Universal Robots PolyScope program: Assem_SubAssem1.urp

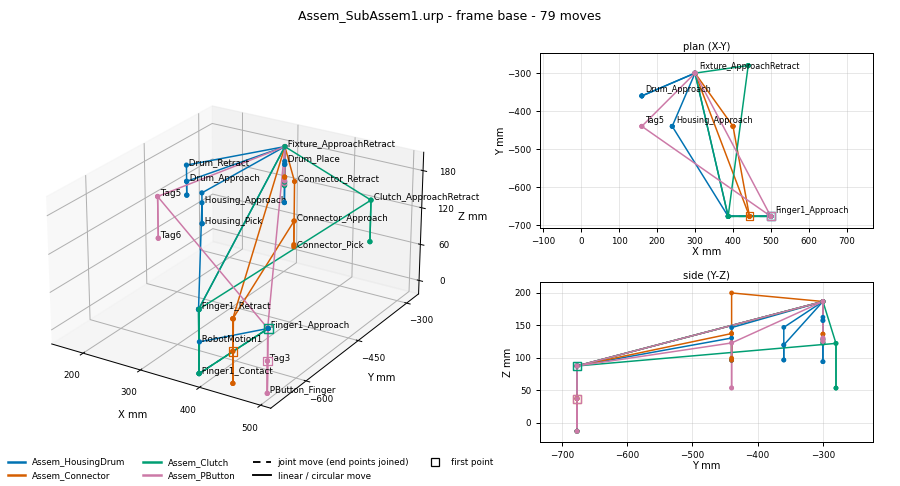
[picture p0: tool path of Assem_SubAssem1.urp in frame base, 79 of 79 moves have a stored position in this frame; points joined in program order, loops and branches not executed]
Program Assem_SubAssem1 (createdIn=3.7.2.40245 lastSavedIn=3.7.2.40245 robotSerialNumber= directory= installation=)
Robot Program (runOnlyOnce=false)
  Call Assem_HousingDrum
  Call Assem_Connector
  Call Assem_Clutch
  Call Assem_PButton
SubProgram -> Assem_HousingDrum
SubProgram -> Assem_Connector
SubProgram -> Assem_Clutch
SubProgram -> Assem_PButton
SubProgram Assem_HousingDrum (keepSynchronizedWithDisk=false trackProgramExecution=true)
  MoveJ speed 120 deg/s, acceleration 360 deg/s^2 (useActiveTCP=false) tcp=TCP_1; feature=Base
    Waypoint Finger1_Approach: TCP in base x=500.448 y=-677.024 z=87.412 mm, rx=-2.2214 ry=2.2214 rz=0 rad; joints [-44.419, -144.242, -45.363, -80.394, 90, -44.419] deg; flange x=500.447 y=-677.022 z=245.817 mm, rx=-2.2214 ry=2.2214 rz=0 rad
  Script: rq_activate_and_wait()
  URCap Gripper (Robotiq_Grippers, Robotiq Inc.) dataModel(position=25, force=50, speed=50, blocking=true, positionInDouble=25.0, forceInDouble=50.0, speedInDouble=50.0)
  MoveL speed 250 mm/s, acceleration 5000 mm/s^2 (useActiveTCP=false) tcp=TCP_1; feature=Base
    Waypoint RobotMotion1: TCP in base x=388.248 y=-677.024 z=37.407 mm, rx=2.2214 ry=-2.2214 rz=0 rad; joints [-50.333, -136.868, -66.833, -66.298, 90, -50.333] deg; flange x=388.247 y=-677.023 z=195.812 mm, rx=2.2214 ry=-2.2214 rz=0 rad
  Set DigitalOutput pin=config_out[0]; digitalValue=1
  MoveL speed 250 mm/s, acceleration 5000 mm/s^2 (useActiveTCP=false) tcp=TCP_1; feature=Base
    Waypoint Finger1_Contact: TCP in base x=387.249 y=-677.025 z=-12.589 mm, rx=-2.2214 ry=2.2214 rz=-0.0001 rad; joints [-50.391, -140.03, -68.963, -61.003, 90, -50.39] deg; flange x=387.242 y=-677.017 z=145.816 mm, rx=-2.2214 ry=2.2214 rz=-0.0001 rad
  Set DigitalOutput pin=config_out[0]; digitalValue=0
  Wait Sleep waitTime=1
  MoveL speed 250 mm/s, acceleration 5000 mm/s^2 (useActiveTCP=false) tcp=TCP_1; feature=Base
    Waypoint Finger1_Retract: TCP in base x=387.248 y=-677.024 z=87.414 mm, rx=-2.2214 ry=2.2214 rz=0 rad; joints [-50.39, -134.151, -63.976, -71.872, 90, -50.39] deg; flange x=387.246 y=-677.022 z=245.819 mm, rx=-2.2214 ry=2.2214 rz=0 rad
  MoveL speed 250 mm/s, acceleration 5000 mm/s^2 (useActiveTCP=false) tcp=TCP_1; feature=Base
    Waypoint Housing_Approach: TCP in base x=240 y=-440 z=130.253 mm, rx=2.2214 ry=-2.2214 rz=0 rad; joints [-45.965, -95.978, -114.162, -59.858, 90, -45.965] deg; flange x=239.997 y=-439.996 z=288.658 mm, rx=2.2214 ry=-2.2214 rz=0 rad
  MoveL speed 250 mm/s, acceleration 5000 mm/s^2 (useActiveTCP=false) tcp=TCP_1; feature=Base
    Waypoint Housing_Pick: TCP in base x=240 y=-440 z=96.255 mm, rx=-2.2214 ry=2.2214 rz=-0.0001 rad; joints [-45.965, -98.735, -116.867, -54.395, 90, -45.965] deg; flange x=239.994 y=-439.994 z=254.66 mm, rx=-2.2214 ry=2.2214 rz=-0.0001 rad
  URCap Gripper (Robotiq_Grippers, Robotiq Inc.) dataModel(position=80, force=50, speed=50, blocking=true, positionInDouble=80.0, forceInDouble=50.0, speedInDouble=50.0)
  MoveL speed 250 mm/s, acceleration 5000 mm/s^2 (useActiveTCP=false) tcp=TCP_1; feature=Base
    Waypoint RobotMotion2: TCP in base x=240 y=-440 z=96.257 mm, rx=2.2214 ry=-2.2214 rz=0.0001 rad; joints [-45.965, -98.735, -116.866, -54.397, 90, -45.965] deg; flange x=239.996 y=-439.995 z=254.662 mm, rx=2.2214 ry=-2.2214 rz=0.0001 rad
  MoveL speed 250 mm/s, acceleration 5000 mm/s^2 (useActiveTCP=false) tcp=TCP_1; feature=Base
    Waypoint Housing_Retract: TCP in base x=240 y=-439.999 z=146.257 mm, rx=2.2214 ry=-2.2214 rz=0.0001 rad; joints [-45.965, -94.842, -112.761, -62.393, 90, -45.965] deg; flange x=239.994 y=-439.993 z=304.662 mm, rx=2.2214 ry=-2.2214 rz=0.0001 rad
  MoveL speed 250 mm/s, acceleration 5000 mm/s^2 (useActiveTCP=false) tcp=TCP_1; feature=Base
    Waypoint Fixture_ApproachRetract: TCP in base x=299.997 y=-299.998 z=186.263 mm, rx=-2.2214 ry=2.2214 rz=-0.0002 rad; joints [-26.687, -81.35, -119.315, -69.329, 89.999, -26.687] deg; flange x=299.983 y=-299.987 z=344.668 mm, rx=-2.2214 ry=2.2214 rz=-0.0002 rad
  MoveL speed 250 mm/s, acceleration 5000 mm/s^2 (useActiveTCP=false) tcp=TCP_1; feature=Base
    Waypoint Housing_Place: TCP in base x=300 y=-300 z=94.01 mm, rx=-2.2214 ry=2.2214 rz=-0.0001 rad; joints [-26.687, -88.56, -128.317, -53.117, 89.999, -26.687] deg; flange x=299.989 y=-299.991 z=252.415 mm, rx=-2.2214 ry=2.2214 rz=-0.0001 rad
  URCap Gripper (Robotiq_Grippers, Robotiq Inc.) dataModel(position=25, force=50, speed=50, blocking=true, positionInDouble=25.0, forceInDouble=50.0, speedInDouble=50.0)
  MoveL speed 250 mm/s, acceleration 5000 mm/s^2 (useActiveTCP=false) tcp=TCP_1; feature=Base
    Waypoint RobotMotion3: TCP in base x=300.001 y=-300 z=94.012 mm, rx=-2.2214 ry=2.2214 rz=-0.0002 rad; joints [-26.687, -88.56, -128.317, -53.117, 89.999, -26.687] deg; flange x=299.988 y=-299.991 z=252.417 mm, rx=-2.2214 ry=2.2214 rz=-0.0002 rad
  MoveL speed 250 mm/s, acceleration 5000 mm/s^2 (useActiveTCP=false) tcp=TCP_1; feature=Base
    Waypoint Fixture_ApproachRetract: TCP in base x=299.997 y=-299.998 z=186.263 mm, rx=-2.2214 ry=2.2214 rz=-0.0002 rad; joints [-26.687, -81.35, -119.315, -69.329, 89.999, -26.687] deg; flange x=299.983 y=-299.987 z=344.668 mm, rx=-2.2214 ry=2.2214 rz=-0.0002 rad
  MoveL speed 250 mm/s, acceleration 5000 mm/s^2 (useActiveTCP=false) tcp=TCP_1; feature=Base
    Waypoint Drum_Approach: TCP in base x=160 y=-360 z=119.602 mm, rx=-2.2214 ry=2.2214 rz=-0.0002 rad; joints [-46.261, -81.439, -130.102, -58.452, 90.001, -46.261] deg; flange x=159.987 y=-359.99 z=278.007 mm, rx=-2.2214 ry=2.2214 rz=-0.0002 rad
  URCap Gripper (Robotiq_Grippers, Robotiq Inc.) dataModel(position=100, force=50, speed=50, blocking=true, positionInDouble=100.0, forceInDouble=50.0, speedInDouble=50.0)
  MoveL speed 250 mm/s, acceleration 5000 mm/s^2 (useActiveTCP=false) tcp=TCP_1; feature=Base
    Waypoint RobotMotion4: TCP in base x=160 y=-360 z=119.604 mm, rx=-2.2214 ry=2.2214 rz=0 rad; joints [-46.26, -81.442, -130.099, -58.459, 90, -46.26] deg; flange x=159.999 y=-359.999 z=278.009 mm, rx=-2.2214 ry=2.2214 rz=0 rad
  MoveL speed 250 mm/s, acceleration 5000 mm/s^2 (useActiveTCP=false) tcp=TCP_1; feature=Base
    Waypoint Drum_Pick: TCP in base x=160 y=-360 z=96.603 mm, rx=-2.2214 ry=2.2214 rz=0 rad; joints [-46.26, -83.73, -132.237, -54.031, 90, -46.26] deg; flange x=159.999 y=-359.999 z=255.008 mm, rx=-2.2214 ry=2.2214 rz=0 rad
  URCap Gripper (Robotiq_Grippers, Robotiq Inc.) dataModel(position=90, force=50, speed=50, blocking=true, positionInDouble=90.0, forceInDouble=50.0, speedInDouble=50.0)
  MoveL speed 250 mm/s, acceleration 5000 mm/s^2 (useActiveTCP=false) tcp=TCP_1; feature=Base
    Waypoint RobotMotion5: TCP in base x=160 y=-360 z=96.605 mm, rx=-2.2214 ry=2.2214 rz=0 rad; joints [-46.26, -83.73, -132.237, -54.031, 90, -46.26] deg; flange x=159.998 y=-359.998 z=255.01 mm, rx=-2.2214 ry=2.2214 rz=0 rad
  MoveL speed 250 mm/s, acceleration 5000 mm/s^2 (useActiveTCP=false) tcp=TCP_1; feature=Base
    Waypoint Drum_Retract: TCP in base x=160 y=-360 z=146.603 mm, rx=-2.2214 ry=2.2214 rz=0 rad; joints [-46.26, -79.175, -127.379, -63.445, 90, -46.26] deg; flange x=159.998 y=-359.998 z=305.008 mm, rx=-2.2214 ry=2.2214 rz=0 rad
  MoveL speed 250 mm/s, acceleration 5000 mm/s^2 (useActiveTCP=false) tcp=TCP_1; feature=Base
    Waypoint Fixture_ApproachRetract: TCP in base x=299.997 y=-299.998 z=186.263 mm, rx=-2.2214 ry=2.2214 rz=-0.0002 rad; joints [-26.687, -81.35, -119.315, -69.329, 89.999, -26.687] deg; flange x=299.983 y=-299.987 z=344.668 mm, rx=-2.2214 ry=2.2214 rz=-0.0002 rad
  MoveL speed 250 mm/s, acceleration 5000 mm/s^2 (useActiveTCP=false) tcp=TCP_1; feature=Base
    Waypoint Drum_Align: TCP in base x=299.997 y=-299.998 z=186.263 mm, rx=1.0745 ry=-2.9521 rz=0.0002 rad; joints [-26.684, -81.35, -119.314, -69.332, 89.995, 23.316] deg; flange x=299.996 y=-299.98 z=344.668 mm, rx=1.0745 ry=-2.9521 rz=0.0002 rad
  MoveL speed 250 mm/s, acceleration 5000 mm/s^2 (useActiveTCP=false) tcp=TCP_1; feature=Base
    Waypoint Drum_Place: TCP in base x=300 y=-300 z=162.113 mm, rx=-1.0745 ry=2.9521 rz=0 rad; joints [-26.688, -82.813, -121.912, -65.274, 90, 23.312] deg; flange x=299.998 y=-299.999 z=320.518 mm, rx=-1.0745 ry=2.9521 rz=0 rad
  MoveL speed 250 mm/s, acceleration 5000 mm/s^2 (useActiveTCP=false) tcp=TCP_1; feature=Base
    Waypoint Drum_Insert: TCP in base x=300 y=-300 z=157.114 mm, rx=3.0671 ry=0.68 rz=0 rad; joints [-26.688, -83.151, -122.43, -64.418, 90, -141.688] deg; flange x=299.997 y=-299.999 z=315.519 mm, rx=3.0671 ry=0.68 rz=0 rad
  URCap Gripper (Robotiq_Grippers, Robotiq Inc.) dataModel(position=100, force=50, speed=50, blocking=true, positionInDouble=100.0, forceInDouble=50.0, speedInDouble=50.0)
  MoveL speed 250 mm/s, acceleration 5000 mm/s^2 (useActiveTCP=false) tcp=TCP_1; feature=Base
    Waypoint RobotMotion6: TCP in base x=299.999 y=-299.999 z=157.115 mm, rx=3.0671 ry=0.68 rz=0 rad; joints [-26.688, -83.151, -122.43, -64.418, 90, -141.688] deg; flange x=299.997 y=-299.998 z=315.52 mm, rx=3.0671 ry=0.68 rz=0 rad
  MoveL speed 250 mm/s, acceleration 5000 mm/s^2 (useActiveTCP=false) tcp=TCP_1; feature=Base
    Waypoint Fixture_ApproachRetract: TCP in base x=299.997 y=-299.998 z=186.263 mm, rx=-2.2214 ry=2.2214 rz=-0.0002 rad; joints [-26.687, -81.35, -119.315, -69.329, 89.999, -26.687] deg; flange x=299.983 y=-299.987 z=344.668 mm, rx=-2.2214 ry=2.2214 rz=-0.0002 rad
  MoveL speed 250 mm/s, acceleration 5000 mm/s^2 (useActiveTCP=false) tcp=TCP_1; feature=Base
    Waypoint Finger1_Retract: TCP in base x=387.248 y=-677.024 z=87.414 mm, rx=-2.2214 ry=2.2214 rz=0 rad; joints [-50.39, -134.151, -63.976, -71.872, 90, -50.39] deg; flange x=387.246 y=-677.022 z=245.819 mm, rx=-2.2214 ry=2.2214 rz=0 rad
  URCap Gripper (Robotiq_Grippers, Robotiq Inc.) dataModel(position=25, force=50, speed=50, blocking=true, positionInDouble=25.0, forceInDouble=50.0, speedInDouble=50.0)
  MoveL speed 250 mm/s, acceleration 5000 mm/s^2 (useActiveTCP=false) tcp=TCP_1; feature=Base
    Waypoint RobotMotion7: TCP in base x=388.249 y=-677.024 z=87.418 mm, rx=2.2214 ry=-2.2214 rz=0 rad; joints [-50.333, -134.223, -63.846, -71.929, 90, -50.333] deg; flange x=388.246 y=-677.022 z=245.823 mm, rx=2.2214 ry=-2.2214 rz=0 rad
  MoveL speed 250 mm/s, acceleration 5000 mm/s^2 (useActiveTCP=false) tcp=TCP_1; feature=Base
    Waypoint Finger1_Contact: TCP in base x=387.249 y=-677.025 z=-12.589 mm, rx=-2.2214 ry=2.2214 rz=-0.0001 rad; joints [-50.391, -140.03, -68.963, -61.003, 90, -50.39] deg; flange x=387.242 y=-677.017 z=145.816 mm, rx=-2.2214 ry=2.2214 rz=-0.0001 rad
  Set DigitalOutput pin=config_out[0]; digitalValue=1
  Wait Sleep waitTime=1
  MoveJ speed 120 deg/s, acceleration 360 deg/s^2 (useActiveTCP=false) tcp=TCP_1; feature=Base
    Waypoint Finger1_Approach: TCP in base x=500.448 y=-677.024 z=87.412 mm, rx=-2.2214 ry=2.2214 rz=0 rad; joints [-44.419, -144.242, -45.363, -80.394, 90, -44.419] deg; flange x=500.447 y=-677.022 z=245.817 mm, rx=-2.2214 ry=2.2214 rz=0 rad
SubProgram Assem_Connector (keepSynchronizedWithDisk=false trackProgramExecution=true)
  MoveL speed 250 mm/s, acceleration 5000 mm/s^2 (useActiveTCP=false) tcp=TCP_1; feature=Base
    Waypoint Finger2_Approach: TCP in base x=443.348 y=-677.023 z=37.402 mm, rx=-2.2214 ry=2.2214 rz=0 rad; joints [-47.301, -140.975, -59.111, -69.913, 90, -47.301] deg; flange x=443.348 y=-677.023 z=195.807 mm, rx=-2.2214 ry=2.2214 rz=0 rad
  MoveL speed 250 mm/s, acceleration 5000 mm/s^2 (useActiveTCP=false) tcp=TCP_1; feature=Base
    Waypoint Finger2_Contact: TCP in base x=443.348 y=-677.023 z=-12.6 mm, rx=2.2214 ry=-2.2214 rz=0 rad; joints [-47.3, -143.968, -61.249, -64.783, 90, -47.3] deg; flange x=443.348 y=-677.023 z=145.805 mm, rx=2.2214 ry=-2.2214 rz=0 rad
  Set DigitalOutput pin=config_out[0]; digitalValue=0
  Wait Sleep waitTime=1
  MoveL speed 250 mm/s, acceleration 5000 mm/s^2 (useActiveTCP=false) tcp=TCP_1; feature=Base
    Waypoint Finger2_Retract: TCP in base x=443.347 y=-677.023 z=87.404 mm, rx=-2.2214 ry=2.2214 rz=0 rad; joints [-47.301, -138.599, -55.894, -75.506, 90, -47.301] deg; flange x=443.346 y=-677.022 z=245.809 mm, rx=-2.2214 ry=2.2214 rz=0 rad
  MoveL speed 250 mm/s, acceleration 5000 mm/s^2 (useActiveTCP=false) tcp=TCP_1; feature=Base
    Waypoint Connector_Approach: TCP in base x=400 y=-440 z=137.121 mm, rx=-2.2214 ry=2.2214 rz=0 rad; joints [-34.772, -133.787, -57.117, 100.904, -90, 145.228] deg; flange x=400 y=-440 z=295.526 mm, rx=-2.2214 ry=2.2214 rz=0 rad
  MoveL speed 250 mm/s, acceleration 5000 mm/s^2 (useActiveTCP=false) tcp=TCP_1; feature=Base
    Waypoint RobotMotion1: TCP in base x=400 y=-440 z=137.127 mm, rx=-2.2214 ry=2.2214 rz=0 rad; joints [-34.772, -133.786, -57.117, 100.904, -90, 145.228] deg; flange x=399.998 y=-439.999 z=295.532 mm, rx=-2.2214 ry=2.2214 rz=0 rad
  MoveL speed 250 mm/s, acceleration 5000 mm/s^2 (useActiveTCP=false) tcp=TCP_1; feature=Base
    Waypoint Connector_Pick: TCP in base x=400 y=-440 z=96.11 mm, rx=-2.2214 ry=2.2214 rz=0 rad; joints [-34.772, -135.283, -60.612, 105.896, -90, 145.228] deg; flange x=399.999 y=-439.999 z=254.515 mm, rx=-2.2214 ry=2.2214 rz=0 rad
  URCap Gripper (Robotiq_Grippers, Robotiq Inc.) dataModel(position=85, force=50, speed=50, blocking=true, positionInDouble=85.0, forceInDouble=50.0, speedInDouble=50.0)
  MoveL speed 250 mm/s, acceleration 5000 mm/s^2 (useActiveTCP=false) tcp=TCP_1; feature=Base
    Waypoint RobotMotion2: TCP in base x=400.001 y=-440 z=99.381 mm, rx=-2.2214 ry=2.2214 rz=0 rad; joints [-34.772, -135.146, -60.363, 105.51, -90, 145.228] deg; flange x=399.998 y=-439.998 z=257.786 mm, rx=-2.2214 ry=2.2214 rz=0 rad
  MoveL speed 250 mm/s, acceleration 5000 mm/s^2 (useActiveTCP=false) tcp=TCP_1; feature=Base
    Waypoint Connector_Retract: TCP in base x=399.999 y=-439.999 z=199.381 mm, rx=-2.2214 ry=2.2214 rz=0 rad; joints [-34.772, -132.555, -50.102, 92.658, -90, 145.228] deg; flange x=399.996 y=-439.997 z=357.786 mm, rx=-2.2214 ry=2.2214 rz=0 rad
  MoveL speed 250 mm/s, acceleration 5000 mm/s^2 (useActiveTCP=false) tcp=TCP_1; feature=Base
    Waypoint Fixture_ApproachRetract: TCP in base x=299.997 y=-299.998 z=186.263 mm, rx=-2.2214 ry=2.2214 rz=-0.0002 rad; joints [-26.687, -107.809, -90.446, 108.261, -89.999, 153.313] deg; flange x=299.983 y=-299.987 z=344.668 mm, rx=-2.2214 ry=2.2214 rz=-0.0002 rad
  MoveL speed 250 mm/s, acceleration 5000 mm/s^2 (useActiveTCP=false) tcp=TCP_1; feature=Base
    Waypoint Connector_Place: TCP in base x=300.002 y=-300.001 z=136.264 mm, rx=-2.2214 ry=2.2214 rz=-0.0002 rad; joints [-26.687, -110.306, -94.864, 115.177, -89.999, 153.313] deg; flange x=299.987 y=-299.99 z=294.669 mm, rx=-2.2214 ry=2.2214 rz=-0.0002 rad
  URCap Gripper (Robotiq_Grippers, Robotiq Inc.) dataModel(position=100, force=50, speed=50, blocking=true, positionInDouble=100.0, forceInDouble=50.0, speedInDouble=50.0)
  MoveL speed 250 mm/s, acceleration 5000 mm/s^2 (useActiveTCP=false) tcp=TCP_1; feature=Base
    Waypoint RobotMotion3: TCP in base x=300.002 y=-300.001 z=136.267 mm, rx=-2.2214 ry=2.2214 rz=-0.0002 rad; joints [-26.687, -110.305, -94.864, 115.177, -89.999, 153.313] deg; flange x=299.986 y=-299.989 z=294.672 mm, rx=-2.2214 ry=2.2214 rz=-0.0002 rad
  MoveL speed 250 mm/s, acceleration 5000 mm/s^2 (useActiveTCP=false) tcp=TCP_1; feature=Base
    Waypoint Fixture_ApproachRetract: TCP in base x=299.997 y=-299.998 z=186.263 mm, rx=-2.2214 ry=2.2214 rz=-0.0002 rad; joints [-26.687, -107.809, -90.446, 108.261, -89.999, 153.313] deg; flange x=299.983 y=-299.987 z=344.668 mm, rx=-2.2214 ry=2.2214 rz=-0.0002 rad
  MoveL speed 250 mm/s, acceleration 5000 mm/s^2 (useActiveTCP=false) tcp=TCP_1; feature=Base
    Waypoint Finger2_Retract: TCP in base x=443.347 y=-677.023 z=87.404 mm, rx=-2.2214 ry=2.2214 rz=0 rad; joints [0, 0, 0, 0, 0, 0] deg; flange x=443.346 y=-677.022 z=245.809 mm, rx=-2.2214 ry=2.2214 rz=0 rad
  URCap Gripper (Robotiq_Grippers, Robotiq Inc.) dataModel(position=25, force=50, speed=50, blocking=true, positionInDouble=25.0, forceInDouble=50.0, speedInDouble=50.0)
  MoveL speed 250 mm/s, acceleration 5000 mm/s^2 (useActiveTCP=false) tcp=TCP_1; feature=Base
    Waypoint RobotMotion4: TCP in base x=444.348 y=-677.023 z=87.407 mm, rx=-2.2214 ry=2.2214 rz=0 rad; joints [0, 0, 0, 0, 0, 0] deg; flange x=444.346 y=-677.022 z=245.812 mm, rx=-2.2214 ry=2.2214 rz=0 rad
  MoveL speed 250 mm/s, acceleration 5000 mm/s^2 (useActiveTCP=false) tcp=TCP_1; feature=Base
    Waypoint Finger2_Contact: TCP in base x=443.348 y=-677.023 z=-12.6 mm, rx=2.2214 ry=-2.2214 rz=0 rad; joints [0, 0, 0, 0, 0, 0] deg; flange x=443.348 y=-677.023 z=145.805 mm, rx=2.2214 ry=-2.2214 rz=0 rad
  Set DigitalOutput pin=config_out[0]; digitalValue=1
  Wait Sleep waitTime=1
  MoveL speed 250 mm/s, acceleration 5000 mm/s^2 (useActiveTCP=false) tcp=TCP_1; feature=Base
    Waypoint Finger2_Approach: TCP in base x=443.348 y=-677.023 z=37.402 mm, rx=-2.2214 ry=2.2214 rz=0 rad; joints [0, 0, 0, 0, 0, 0] deg; flange x=443.348 y=-677.023 z=195.807 mm, rx=-2.2214 ry=2.2214 rz=0 rad
SubProgram Assem_Clutch (keepSynchronizedWithDisk=false trackProgramExecution=true)
  MoveL speed 250 mm/s, acceleration 5000 mm/s^2 (useActiveTCP=false) tcp=TCP_1; feature=Base
    Waypoint Finger1_Approach: TCP in base x=500.448 y=-677.024 z=87.412 mm, rx=-2.2214 ry=2.2214 rz=0 rad; joints [0, 0, 0, 0, 0, 0] deg; flange x=500.447 y=-677.022 z=245.817 mm, rx=-2.2214 ry=2.2214 rz=0 rad
  MoveL speed 250 mm/s, acceleration 5000 mm/s^2 (useActiveTCP=false) tcp=TCP_1; feature=Base
    Waypoint Finger1_Contact: TCP in base x=387.249 y=-677.025 z=-12.589 mm, rx=-2.2214 ry=2.2214 rz=-0.0001 rad; joints [0, 0, 0, 0, 0, 0] deg; flange x=387.242 y=-677.017 z=145.816 mm, rx=-2.2214 ry=2.2214 rz=-0.0001 rad
  Set DigitalOutput pin=config_out[0]; digitalValue=0
  Wait Sleep waitTime=1
  MoveL speed 250 mm/s, acceleration 5000 mm/s^2 (useActiveTCP=false) tcp=TCP_1; feature=Base
    Waypoint Finger1_Retract: TCP in base x=387.248 y=-677.024 z=87.414 mm, rx=-2.2214 ry=2.2214 rz=0 rad; joints [0, 0, 0, 0, 0, 0] deg; flange x=387.246 y=-677.022 z=245.819 mm, rx=-2.2214 ry=2.2214 rz=0 rad
  MoveL speed 250 mm/s, acceleration 5000 mm/s^2 (useActiveTCP=false) tcp=TCP_1; feature=Base
    Waypoint Clutch_ApproachRetract: TCP in base x=440 y=-280 z=122.051 mm, rx=-2.2214 ry=2.2214 rz=0 rad; joints [-17.663, -123.732, -76.54, 110.273, -90, 162.337] deg; flange x=440 y=-280 z=280.456 mm, rx=-2.2214 ry=2.2214 rz=0 rad
  MoveL speed 250 mm/s, acceleration 5000 mm/s^2 (useActiveTCP=false) tcp=TCP_1; feature=Base
    Waypoint Clutch_Pick: TCP in base x=440 y=-280 z=53.553 mm, rx=-2.2214 ry=2.2214 rz=0 rad; joints [-17.663, -127.625, -80.942, 118.568, -90, 162.337] deg; flange x=440 y=-280 z=211.958 mm, rx=-2.2214 ry=2.2214 rz=0 rad
  URCap Gripper (Robotiq_Grippers, Robotiq Inc.) dataModel(position=88, force=50, speed=50, blocking=true, positionInDouble=88.0, forceInDouble=50.0, speedInDouble=50.0)
  MoveL speed 250 mm/s, acceleration 5000 mm/s^2 (useActiveTCP=false) tcp=TCP_1; feature=Base
    Waypoint RobotMotion1: TCP in base x=440 y=-280 z=53.554 mm, rx=-2.2214 ry=2.2214 rz=0 rad; joints [-17.663, -127.625, -80.942, 118.568, -90, 162.337] deg; flange x=439.999 y=-280 z=211.959 mm, rx=-2.2214 ry=2.2214 rz=0 rad
  MoveL speed 250 mm/s, acceleration 5000 mm/s^2 (useActiveTCP=false) tcp=TCP_1; feature=Base
    Waypoint Clutch_ApproachRetract: TCP in base x=440 y=-280 z=122.051 mm, rx=-2.2214 ry=2.2214 rz=0 rad; joints [-17.663, -123.732, -76.54, 110.273, -90, 162.337] deg; flange x=440 y=-280 z=280.456 mm, rx=-2.2214 ry=2.2214 rz=0 rad
  MoveL speed 250 mm/s, acceleration 5000 mm/s^2 (useActiveTCP=false) tcp=TCP_1; feature=Base
    Waypoint Fixture_ApproachRetract: TCP in base x=299.997 y=-299.998 z=186.263 mm, rx=-2.2214 ry=2.2214 rz=-0.0002 rad; joints [-26.687, -107.809, -90.446, 108.261, -89.999, 153.313] deg; flange x=299.983 y=-299.987 z=344.668 mm, rx=-2.2214 ry=2.2214 rz=-0.0002 rad
  MoveL speed 250 mm/s, acceleration 5000 mm/s^2 (useActiveTCP=false) tcp=TCP_1; feature=Base
    Waypoint Clutch_Place: TCP in base x=300.003 y=-300.002 z=123.266 mm, rx=-2.2214 ry=2.2214 rz=-0.0002 rad; joints [-26.687, -111.079, -95.875, 116.961, -89.999, 153.313] deg; flange x=299.987 y=-299.99 z=281.671 mm, rx=-2.2214 ry=2.2214 rz=-0.0002 rad
  URCap Gripper (Robotiq_Grippers, Robotiq Inc.) dataModel(position=75, force=50, speed=50, blocking=true, positionInDouble=75.0, forceInDouble=50.0, speedInDouble=50.0)
  MoveL speed 250 mm/s, acceleration 5000 mm/s^2 (useActiveTCP=false) tcp=TCP_1; feature=Base
    Waypoint RobotMotion2: TCP in base x=300.003 y=-300.002 z=123.267 mm, rx=-2.2214 ry=2.2214 rz=-0.0002 rad; joints [-26.687, -111.079, -95.875, 116.961, -89.999, 153.313] deg; flange x=299.987 y=-299.99 z=281.672 mm, rx=-2.2214 ry=2.2214 rz=-0.0002 rad
  MoveL speed 250 mm/s, acceleration 5000 mm/s^2 (useActiveTCP=false) tcp=TCP_1; feature=Base
    Waypoint Clutch_PushRetract: TCP in base x=300.003 y=-300.001 z=128.267 mm, rx=-2.2214 ry=2.2214 rz=-0.0002 rad; joints [-26.687, -110.776, -95.493, 116.276, -89.999, 153.313] deg; flange x=299.987 y=-299.99 z=286.672 mm, rx=-2.2214 ry=2.2214 rz=-0.0002 rad
  URCap Gripper (Robotiq_Grippers, Robotiq Inc.) dataModel(position=100, force=50, speed=50, blocking=true, positionInDouble=100.0, forceInDouble=50.0, speedInDouble=50.0)
  MoveL speed 250 mm/s, acceleration 5000 mm/s^2 (useActiveTCP=false) tcp=TCP_1; feature=Base
    Waypoint RobotMotion3: TCP in base x=300.003 y=-300.001 z=128.268 mm, rx=-2.2214 ry=2.2214 rz=-0.0002 rad; joints [-26.687, -110.775, -95.493, 116.276, -89.999, 153.313] deg; flange x=299.986 y=-299.99 z=286.673 mm, rx=-2.2214 ry=2.2214 rz=-0.0002 rad
  MoveL speed 250 mm/s, acceleration 5000 mm/s^2 (useActiveTCP=false) tcp=TCP_1; feature=Base
    Waypoint Clutch_Push: TCP in base x=300.003 y=-300.002 z=122.11 mm, rx=-2.2214 ry=2.2214 rz=-0.0002 rad; joints [-26.687, -111.15, -95.962, 117.12, -89.999, 153.313] deg; flange x=299.987 y=-299.99 z=280.515 mm, rx=-2.2214 ry=2.2214 rz=-0.0002 rad
  MoveL speed 250 mm/s, acceleration 5000 mm/s^2 (useActiveTCP=false) tcp=TCP_1; feature=Base
    Waypoint Fixture_ApproachRetract: TCP in base x=299.997 y=-299.998 z=186.263 mm, rx=-2.2214 ry=2.2214 rz=-0.0002 rad; joints [-26.687, -107.809, -90.446, 108.261, -89.999, 153.313] deg; flange x=299.983 y=-299.987 z=344.668 mm, rx=-2.2214 ry=2.2214 rz=-0.0002 rad
  MoveL speed 250 mm/s, acceleration 5000 mm/s^2 (useActiveTCP=false) tcp=TCP_1; feature=Base
    Waypoint Finger1_Retract: TCP in base x=387.248 y=-677.024 z=87.414 mm, rx=-2.2214 ry=2.2214 rz=0 rad; joints [0, 0, 0, 0, 0, 0] deg; flange x=387.246 y=-677.022 z=245.819 mm, rx=-2.2214 ry=2.2214 rz=0 rad
  URCap Gripper (Robotiq_Grippers, Robotiq Inc.) dataModel(position=25, force=50, speed=50, blocking=true, positionInDouble=25.0, forceInDouble=50.0, speedInDouble=50.0)
  MoveL speed 250 mm/s, acceleration 5000 mm/s^2 (useActiveTCP=false) tcp=TCP_1; feature=Base
    Waypoint RobotMotion4: TCP in base x=388.249 y=-677.024 z=87.425 mm, rx=-2.2214 ry=2.2214 rz=-0.0001 rad; joints [0, 0, 0, 0, 0, 0] deg; flange x=388.244 y=-677.021 z=245.83 mm, rx=-2.2214 ry=2.2214 rz=-0.0001 rad
  MoveL speed 250 mm/s, acceleration 5000 mm/s^2 (useActiveTCP=false) tcp=TCP_1; feature=Base
    Waypoint Finger1_Contact: TCP in base x=387.249 y=-677.025 z=-12.589 mm, rx=-2.2214 ry=2.2214 rz=-0.0001 rad; joints [0, 0, 0, 0, 0, 0] deg; flange x=387.242 y=-677.017 z=145.816 mm, rx=-2.2214 ry=2.2214 rz=-0.0001 rad
  Set DigitalOutput pin=config_out[0]; digitalValue=1
  Wait Sleep waitTime=1
  MoveL speed 250 mm/s, acceleration 5000 mm/s^2 (useActiveTCP=false) tcp=TCP_1; feature=Base
    Waypoint Finger1_Approach: TCP in base x=500.448 y=-677.024 z=87.412 mm, rx=-2.2214 ry=2.2214 rz=0 rad; joints [0, 0, 0, 0, 0, 0] deg; flange x=500.447 y=-677.022 z=245.817 mm, rx=-2.2214 ry=2.2214 rz=0 rad
SubProgram Assem_PButton (keepSynchronizedWithDisk=false trackProgramExecution=true)
  MoveL speed 250 mm/s, acceleration 5000 mm/s^2 (useActiveTCP=false) tcp=TCP_1; feature=Base
    Waypoint Tag3: TCP in base x=499.448 y=-677.023 z=37.402 mm, rx=-2.2214 ry=2.2214 rz=0 rad; joints [0, 0, 0, 0, 0, 0] deg; flange x=499.448 y=-677.023 z=195.807 mm, rx=-2.2214 ry=2.2214 rz=0 rad
  MoveL speed 250 mm/s, acceleration 5000 mm/s^2 (useActiveTCP=false) tcp=TCP_1; feature=Base
    Waypoint PButton_Finger: TCP in base x=499.448 y=-677.023 z=-12.6 mm, rx=2.2214 ry=-2.2214 rz=0 rad; joints [0, 0, 0, 0, 0, 0] deg; flange x=499.448 y=-677.023 z=145.805 mm, rx=2.2214 ry=-2.2214 rz=0 rad
  Set DigitalOutput pin=config_out[0]; digitalValue=0
  Wait Sleep waitTime=1
  MoveL speed 250 mm/s, acceleration 5000 mm/s^2 (useActiveTCP=false) tcp=TCP_1; feature=Base
    Waypoint Tag4: TCP in base x=499.448 y=-677.023 z=87.404 mm, rx=-2.2214 ry=2.2214 rz=0 rad; joints [0, 0, 0, 0, 0, 0] deg; flange x=499.447 y=-677.023 z=245.809 mm, rx=-2.2214 ry=2.2214 rz=0 rad
  MoveL speed 250 mm/s, acceleration 5000 mm/s^2 (useActiveTCP=false) tcp=TCP_1; feature=Base
    Waypoint Tag5: TCP in base x=160 y=-440 z=122.703 mm, rx=2.2214 ry=-2.2214 rz=0 rad; joints [-53.475, -116.716, -87.588, 114.304, -90, 126.525] deg; flange x=160 y=-440 z=281.108 mm, rx=2.2214 ry=-2.2214 rz=0 rad
  MoveL speed 250 mm/s, acceleration 5000 mm/s^2 (useActiveTCP=false) tcp=TCP_1; feature=Base
    Waypoint Tag6: TCP in base x=160 y=-440 z=53.705 mm, rx=2.2214 ry=-2.2214 rz=0 rad; joints [-53.475, -121.187, -91.946, 123.133, -90, 126.525] deg; flange x=160 y=-439.999 z=212.11 mm, rx=2.2214 ry=-2.2214 rz=0 rad
  URCap Gripper (Robotiq_Grippers, Robotiq Inc.) dataModel(position=95, force=50, speed=50, blocking=true, positionInDouble=95.0, forceInDouble=50.0, speedInDouble=50.0)
  MoveL speed 250 mm/s, acceleration 5000 mm/s^2 (useActiveTCP=false) tcp=TCP_1; feature=Base
    Waypoint RobotMotion1: TCP in base x=160 y=-440 z=53.706 mm, rx=2.2214 ry=-2.2214 rz=0 rad; joints [-53.475, -121.187, -91.946, 123.133, -90, 126.525] deg; flange x=160 y=-439.999 z=212.111 mm, rx=2.2214 ry=-2.2214 rz=0 rad
  MoveL speed 250 mm/s, acceleration 5000 mm/s^2 (useActiveTCP=false) tcp=TCP_1; feature=Base
    Waypoint Tag5: TCP in base x=160 y=-440 z=122.703 mm, rx=2.2214 ry=-2.2214 rz=0 rad; joints [-53.475, -116.716, -87.588, 114.304, -90, 126.525] deg; flange x=160 y=-440 z=281.108 mm, rx=2.2214 ry=-2.2214 rz=0 rad
  MoveL speed 250 mm/s, acceleration 5000 mm/s^2 (useActiveTCP=false) tcp=TCP_1; feature=Base
    Waypoint Fixture_ApproachRetract: TCP in base x=299.997 y=-299.998 z=186.263 mm, rx=-2.2214 ry=2.2214 rz=-0.0002 rad; joints [-26.687, -107.809, -90.446, 108.261, -89.999, 153.313] deg; flange x=299.983 y=-299.987 z=344.668 mm, rx=-2.2214 ry=2.2214 rz=-0.0002 rad
  MoveL speed 250 mm/s, acceleration 5000 mm/s^2 (useActiveTCP=false) tcp=TCP_1; feature=Base
    Waypoint Tag7: TCP in base x=300.003 y=-300.002 z=125.268 mm, rx=-2.2214 ry=2.2214 rz=-0.0002 rad; joints [-26.687, -110.957, -95.723, 116.687, -89.999, 153.313] deg; flange x=299.987 y=-299.99 z=283.673 mm, rx=-2.2214 ry=2.2214 rz=-0.0002 rad
  URCap Gripper (Robotiq_Grippers, Robotiq Inc.) dataModel(position=75, force=50, speed=50, blocking=true, positionInDouble=75.0, forceInDouble=50.0, speedInDouble=50.0)
  MoveL speed 250 mm/s, acceleration 5000 mm/s^2 (useActiveTCP=false) tcp=TCP_1; feature=Base
    Waypoint RobotMotion2: TCP in base x=300.004 y=-300.001 z=125.27 mm, rx=-2.2214 ry=2.2214 rz=-0.0002 rad; joints [-26.687, -110.956, -95.723, 116.687, -89.999, 153.313] deg; flange x=299.987 y=-299.989 z=283.675 mm, rx=-2.2214 ry=2.2214 rz=-0.0002 rad
  MoveL speed 250 mm/s, acceleration 5000 mm/s^2 (useActiveTCP=false) tcp=TCP_1; feature=Base
    Waypoint Tag8: TCP in base x=300.003 y=-300.001 z=130.269 mm, rx=-2.2214 ry=2.2214 rz=-0.0002 rad; joints [-26.687, -110.656, -95.338, 116.001, -89.999, 153.313] deg; flange x=299.986 y=-299.989 z=288.674 mm, rx=-2.2214 ry=2.2214 rz=-0.0002 rad
  URCap Gripper (Robotiq_Grippers, Robotiq Inc.) dataModel(position=100, force=50, speed=50, blocking=true, positionInDouble=100.0, forceInDouble=50.0, speedInDouble=50.0)
  MoveL speed 250 mm/s, acceleration 5000 mm/s^2 (useActiveTCP=false) tcp=TCP_1; feature=Base
    Waypoint RobotMotion3: TCP in base x=300.003 y=-300 z=130.274 mm, rx=-2.2214 ry=2.2214 rz=-0.0002 rad; joints [-26.687, -110.655, -95.338, 116.001, -89.999, 153.313] deg; flange x=299.985 y=-299.988 z=288.679 mm, rx=-2.2214 ry=2.2214 rz=-0.0002 rad
  MoveL speed 250 mm/s, acceleration 5000 mm/s^2 (useActiveTCP=false) tcp=TCP_1; feature=Base
    Waypoint Tag9: TCP in base x=300.003 y=-300.001 z=127.27 mm, rx=-2.2214 ry=2.2214 rz=-0.0002 rad; joints [-26.687, -110.835, -95.57, 116.413, -89.999, 153.313] deg; flange x=299.986 y=-299.989 z=285.675 mm, rx=-2.2214 ry=2.2214 rz=-0.0002 rad
  MoveL speed 250 mm/s, acceleration 5000 mm/s^2 (useActiveTCP=false) tcp=TCP_1; feature=Base
    Waypoint Fixture_ApproachRetract: TCP in base x=299.997 y=-299.998 z=186.263 mm, rx=-2.2214 ry=2.2214 rz=-0.0002 rad; joints [-26.687, -107.809, -90.446, 108.261, -89.999, 153.313] deg; flange x=299.983 y=-299.987 z=344.668 mm, rx=-2.2214 ry=2.2214 rz=-0.0002 rad
  MoveL speed 250 mm/s, acceleration 5000 mm/s^2 (useActiveTCP=false) tcp=TCP_1; feature=Base
    Waypoint Tag4: TCP in base x=499.448 y=-677.023 z=87.404 mm, rx=-2.2214 ry=2.2214 rz=0 rad; joints [0, 0, 0, 0, 0, 0] deg; flange x=499.447 y=-677.023 z=245.809 mm, rx=-2.2214 ry=2.2214 rz=0 rad
  URCap Gripper (Robotiq_Grippers, Robotiq Inc.) dataModel(position=25, force=50, speed=50, blocking=true, positionInDouble=25.0, forceInDouble=50.0, speedInDouble=50.0)
  MoveL speed 250 mm/s, acceleration 5000 mm/s^2 (useActiveTCP=false) tcp=TCP_1; feature=Base
    Waypoint RobotMotion4: TCP in base x=500.448 y=-677.024 z=87.41 mm, rx=-2.2214 ry=2.2214 rz=0 rad; joints [0, 0, 0, 0, 0, 0] deg; flange x=500.447 y=-677.022 z=245.815 mm, rx=-2.2214 ry=2.2214 rz=0 rad
  MoveL speed 250 mm/s, acceleration 5000 mm/s^2 (useActiveTCP=false) tcp=TCP_1; feature=Base
    Waypoint PButton_Finger: TCP in base x=499.448 y=-677.023 z=-12.6 mm, rx=2.2214 ry=-2.2214 rz=0 rad; joints [0, 0, 0, 0, 0, 0] deg; flange x=499.448 y=-677.023 z=145.805 mm, rx=2.2214 ry=-2.2214 rz=0 rad
  Set DigitalOutput pin=config_out[0]; digitalValue=1
  Wait Sleep waitTime=1
  MoveL speed 250 mm/s, acceleration 5000 mm/s^2 (useActiveTCP=false) tcp=TCP_1; feature=Base
    Waypoint Tag3: TCP in base x=499.448 y=-677.023 z=37.402 mm, rx=-2.2214 ry=2.2214 rz=0 rad; joints [0, 0, 0, 0, 0, 0] deg; flange x=499.448 y=-677.023 z=195.807 mm, rx=-2.2214 ry=2.2214 rz=0 rad
